Yaskawa INFORM job: B-1-08279-80-SUB-R.JBI

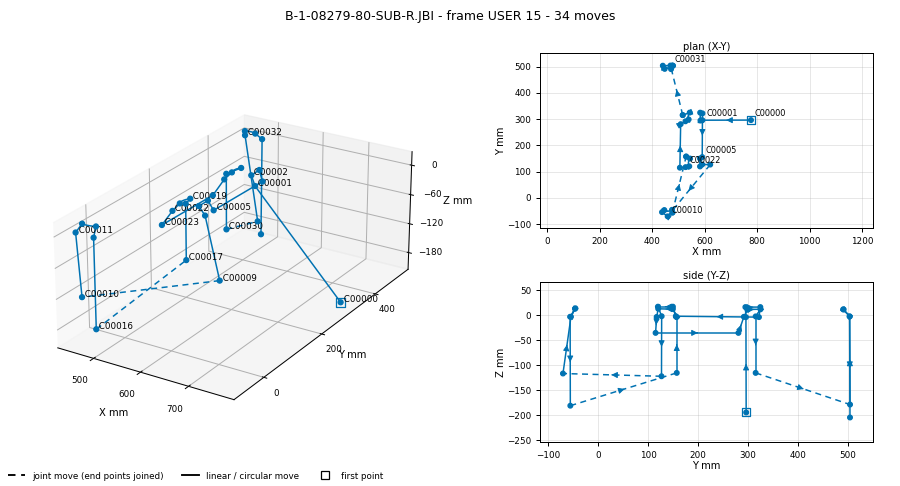
[picture p0: tool path of B-1-08279-80-SUB-R.JBI in frame USER 15, 34 of 38 moves have a stored position in this frame; points joined in program order, loops and branches not executed]
/JOB
//NAME B-1-08279-80-SUB-R
///FOLDERNAME PART_420-08279-80
//POS
///NPOS 38,0,38,0,0,0
///USER 15
///TOOL 4
///POSTYPE USER
///RECTAN
///RCONF 1,0,0,0,0,0,0,0,0,0,0,0,0,0,0,0,0,0,0,0,0,0,0,0
C00000=776.374,296.183,-194.582,-27.8966,11.3058,78.2344
C00001=591.519,295.721,-3.979,-46.5250,6.9320,75.2540
C00002=584.032,294.592,16.068,-46.5264,6.9318,75.2522
C00003=582.978,324.526,16.100,-46.5255,6.9316,75.2547
C00004=591.755,321.720,-3.979,-46.5250,6.9320,75.2540
C00005=590.773,155.478,-2.185,-42.9430,-21.0870,89.6170
C00006=582.419,149.640,16.946,-42.9406,-21.0942,89.6154
C00007=582.419,119.763,16.946,-42.9409,-21.0933,89.6151
C00008=590.773,127.194,-2.185,-42.9430,-21.0870,89.6170
C00009=621.287,126.871,-122.266,-42.9430,-21.0870,89.6170
C00010=459.138,-70.169,-116.763,-6.5599,-44.9783,-116.9691
C00011=437.802,-54.182,-3.282,-6.5590,-44.9790,-116.9690
C00012=446.584,-46.151,12.620,-6.5602,-44.9805,-116.9652
C00013=458.785,-50.245,14.207,-6.5589,-44.9767,-90.5159
C00014=475.749,-45.331,13.727,-6.5562,-44.9812,-55.2611
C00015=477.608,-55.834,-3.282,-6.5580,-44.9790,-55.2560
C00016=477.346,-55.448,-181.107,-6.5568,-44.9787,-55.2555
C00017=529.608,157.384,-115.500,-16.3490,-44.1220,152.7880
C00018=529.609,157.384,-3.682,-16.3490,-44.1220,152.7880
C00019=544.646,149.606,12.241,-12.4955,-45.2511,167.4657
C00020=538.383,134.564,12.293,-16.9646,-44.8177,-161.2144
C00021=541.542,120.323,12.777,-16.5157,-44.7736,-145.3150
C00022=527.621,117.175,-3.669,-16.5140,-44.7720,-151.5720
C00023=505.748,115.031,-35.500,-16.5140,-44.7720,-151.5720
C00024=508.771,280.690,-35.500,3.4420,-44.9790,-154.0720
C00025=527.020,291.566,-3.353,3.4420,-44.9790,-154.0720
C00026=539.186,298.815,10.769,3.4420,-44.9790,-154.0720
C00027=537.624,310.638,11.520,7.8962,-43.2324,176.8590
C00028=543.213,324.833,11.573,15.6683,-44.9794,144.2159
C00029=516.589,315.156,-2.528,16.5470,-44.9790,144.2150
C00030=516.589,315.156,-115.500,16.5470,-44.9790,144.2150
C00031=470.026,503.882,-178.799,28.9267,-36.2202,77.7079
C00032=440.809,503.258,-2.647,28.9260,-36.2220,77.7090
C00033=448.033,491.127,11.426,28.9260,-36.2221,77.7084
C00034=459.382,494.214,11.496,15.7352,-42.8106,71.8260
C00035=472.182,490.167,11.479,13.1194,-43.5301,40.3815
C00036=479.884,503.018,-2.647,12.3290,-43.7170,41.5290
C00037=477.766,503.800,-204.677,12.0366,-43.7829,41.9519
///TOOL 0
///POSTYPE ANGLE
///ANGLE
EC00000=-45.0000
///TOOL 4
EC00001=-45.0000
///TOOL 0
EC00002=-45.0000
EC00003=-45.0000
///TOOL 4
EC00004=-45.0000
EC00005=-45.0000
///TOOL 0
EC00006=-45.0005
EC00007=-45.0005
///TOOL 4
EC00008=-45.0000
EC00009=-45.0000
///TOOL 0
EC00010=-90.0000
///TOOL 4
EC00011=-90.0000
///TOOL 0
EC00012=-90.0000
EC00013=-90.0000
EC00014=-90.0000
///TOOL 4
EC00015=-90.0000
///TOOL 0
EC00016=-90.0000
///TOOL 4
EC00017=-90.0000
EC00018=-90.0000
///TOOL 0
EC00019=-90.0000
EC00020=-90.0000
EC00021=-90.0000
///TOOL 4
EC00022=-90.0000
EC00023=-90.0000
EC00024=-90.0000
EC00025=-90.0000
EC00026=-90.0000
///TOOL 0
EC00027=-90.0000
EC00028=-90.0000
///TOOL 4
EC00029=-90.0000
EC00030=-90.0000
///TOOL 0
EC00031=-90.0000
///TOOL 4
EC00032=-90.0000
///TOOL 0
EC00033=-90.0000
EC00034=-90.0000
EC00035=-90.0000
///TOOL 4
EC00036=-90.0000
///TOOL 0
EC00037=-90.0000
//INST
///DATE 2021/10/29 11:36
///ATTR SC,RW,RJ
////FRAME USER 15
///GROUP1 RB1
///GROUP2 ST3
NOP
'Path Start: PP9
'Warning, the first motion progra
'mmed for this routine was not a
'joint motion
'The following movement has been
'added. Please update your OCTOPU
'Z simulation.
MOVJ C00000 VJ=100.00  +MOVJ EC00000
SMOVL C00001 V=1250.0  +MOVJ EC00001
SMOVL C00002 V=300.0  +MOVJ EC00002
ARCON ASF#(951)
SMOVL C00003 V=8.5  +MOVJ EC00003
ARCOF AEF#(951)
SMOVL C00004 V=1250.0  +MOVJ EC00004
'Path End
'Path Start: PP15
SMOVL C00005 V=1250.0  +MOVJ EC00005
SMOVL C00006 V=300.0  +MOVJ EC00006
ARCON ASF#(951)
SMOVL C00007  +MOVJ EC00007
ARCOF AEF#(951)
SMOVL C00008 V=1250.0  +MOVJ EC00008
SMOVL C00009 V=1250.0  +MOVJ EC00009
'Path End
'Path Start: PP16
MOVJ C00010 VJ=25.00  +MOVJ EC00010
SMOVL C00011 V=1250.0  +MOVJ EC00011
SMOVC C00012 V=300.0  +MOVJ EC00012
ARCON ASF#(951)
SMOVC C00013 V=8.5  +MOVJ EC00013
SMOVC C00014 V=8.5  +MOVJ EC00014
ARCOF AEF#(951)
SMOVL C00015 V=1250.0  +MOVJ EC00015
SMOVL C00016 V=1250.0  +MOVJ EC00016
'Path End
'Path Start: PP19
MOVJ C00017 VJ=100.00  +MOVJ EC00017
SMOVL C00018 V=1250.0  +MOVJ EC00018
SMOVC C00019 V=300.0  +MOVJ EC00019
ARCON ASF#(951)
SMOVC C00020 V=8.5  +MOVJ EC00020
SMOVC C00021 V=8.5  +MOVJ EC00021
ARCOF AEF#(951)
SMOVL C00022 V=1250.0  +MOVJ EC00022
SMOVL C00023 V=1250.0  +MOVJ EC00023
'Path End
'Path Start: PP20
SMOVL C00024 V=1250.0  +MOVJ EC00024
SMOVL C00025 V=1250.0  +MOVJ EC00025
SMOVC C00026 V=300.0  +MOVJ EC00026
ARCON ASF#(951)
SMOVC C00027 V=8.5  +MOVJ EC00027
SMOVC C00028 V=8.5  +MOVJ EC00028
ARCOF AEF#(951)
SMOVL C00029 V=1250.0  +MOVJ EC00029
SMOVL C00030 V=1250.0  +MOVJ EC00030
'Path End
'Path Start: PP22
MOVJ C00031 VJ=100.00  +MOVJ EC00031
SMOVL C00032 V=1250.0  +MOVJ EC00032
SMOVC C00033 V=300.0  +MOVJ EC00033
ARCON ASF#(951)
SMOVC C00034 V=8.5  +MOVJ EC00034
SMOVC C00035 V=8.5  +MOVJ EC00035
ARCOF AEF#(951)
SMOVL C00036 V=1250.0  +MOVJ EC00036
SMOVL C00037 V=1250.0  +MOVJ EC00037
'Path End
END
